Fanuc KAREL source: IO0008.KL

-- PROVISIONAL review KL for V1013-1; original PC SHA256 76a218a3a7aa5ec1410d74cd1b81d8a2d83c8b2c5b9b39cabb4eeab652479859
-- Incomplete behavior may be omitted. Consult companion uncertainty JSON. Do not deploy.
PROGRAM IO0008
%NOLOCKGROUP
-- UNRESOLVED_LOCAL_POOL 5 cells at code offset 13; source declarations unknown
-- DIRECT_LOCAL_WORD_ACCESS alone does not prove INTEGER, REAL, or BOOLEAN
BEGIN
  -- UNRESOLVED_PC offsets 0-18; opcodes 2B,2C,7B
  -- UNRESOLVED_PC offsets 23-30; opcodes 9D,23
  -- UNRESOLVED_PC offsets 35-49; opcodes 2E,22,9D,33,35
  -- UNRESOLVED_PC offsets 54-61; opcodes 9D,23
  -- UNRESOLVED_PC offsets 66-77; opcodes 2E,23
  -- UNRESOLVED_PC offsets 82-97; opcodes 21,19,9D,57,79
  -- UNRESOLVED_PC offsets 102-116; opcodes 21,9D,52,23
  -- UNRESOLVED_PC offsets 126-130; opcodes 7F
  -- UNRESOLVED_PC offsets 135-139; opcodes 27,AA
  -- UNRESOLVED_PC offsets 144-148; opcodes 7F
END IO0008
